FUNCTION_BLOCK IncrementalEncoderWidget
VAR_INPUT
END_VAR
VAR_OUTPUT
END_VAR
VAR_IN_OUT
    ref : IncrementalEncoder;
END_VAR
VAR
	actualStatus : StatusWidget;
END_VAR

actualStatus(text := ref.actualStatus, 
             color := HealthBusyToColor(healthStatus := ref.statuses.healthStatus, 
                                        busyStatus := ref.statuses.busyStatus));

END_FUNCTION_BLOCK

(* stored: Version 1.1.0.1, ProductVersion 3.1.4018.5
   POU IncrementalEncoderWidget: Id {78a49e48-5c49-4e3d-8dd8-83c6fe74bb8c}, SpecialFunc None *)
